Staubli VAL3: N16_AgafarPuntes.pgx

program N16_AgafarPuntes()
  local pointRx l_pAgafarPuntes
  local pointRx l_pAgafarPuntesRapid
begin

  // Anar al punt de la banyera
  if aioGet(aiNumPipeta)==2
    l_pAgafarPuntes=pAgafarPuntes8
  else
    l_pAgafarPuntes=pAgafarPuntes1
  endIf

  l_pAgafarPuntes.trsf.x=l_pAgafarPuntes.trsf.x+nXOffset
  l_pAgafarPuntes.trsf.y=l_pAgafarPuntes.trsf.y+nYOffset
  l_pAgafarPuntes.trsf.z=l_pAgafarPuntes.trsf.z+nZOffset
  l_pAgafarPuntesRapid=l_pAgafarPuntes
  l_pAgafarPuntesRapid.trsf.z=l_pAgafarPuntesRapid.trsf.z+20
  movel(l_pAgafarPuntesRapid,tToolActiva,mLent)
  waitEndMove()
  movel(l_pAgafarPuntes,tToolActiva,mAgafarPuntes)
  waitEndMove()

  bTaskDone=true
end
